// TIA Portal project "Bai 7" (V16)

(* hardware
DEVICE "S7-1200 station_1"  S7-1200 Station
   slot 0: "Rack_0"  S7-1200 Rack  Rack  V1.0
   slot 1: "PLC Powered Off"  CPU 1214C DC/DC/DC  6ES7 214-1AG40-0XB0  V4.2
   slot 2: "DQ 16xRelay_1"  SM 1222 DQ16 x relay  6ES7 222-1HH32-0XB0  V2.0
*)

// ===== PLC "PLC Powered Off"  CPU 1214C DC/DC/DC =====

VAR_GLOBAL   // PLC tag table "Default tag table"
   ""Start"" AT %I0.0 : Bool;
   ""Tag_7"" AT %I0.3 : Bool;
   ""Stop"" AT %I0.1 : Bool;
   ""Quay_DC"" AT %Q9.0 : Bool;
   ""Tag_3"" AT %Q9.1 : Bool;
   ""Tag_4"" AT %Q9.5 : Bool;
   ""Tag_5"" AT %Q9.6 : Bool;
END_VAR